// TIA Portal V19 export
FUNCTION_BLOCK "Prod_O_TODO_Push_ManualOrder"   // FB35, LAD
TITLE = INSERIMENTO MANAULE ORDINE SU LISTA ORDINI DA FARE (HMI -> TODO)
// stored: Access Published, MemoryReserve 100, SetENOAutomatically false
   VAR_INPUT
      Execute : Bool;
      Enable : Bool;
   END_VAR
   VAR_OUTPUT
      Ready : Bool;
      Busy : Bool;
      Done : Bool;
      Error : Bool;
   END_VAR
   VAR
      PPrf_Data_Presence { S7_SetPoint := 'True'} : Bool;
      WriteOrder : Bool;
      Prg { S7_SetPoint := 'True'} : "PPrf_Data";
      PPrf_Get { S7_SetPoint := 'True'} : "GetPrg";
      TON_Timeout { S7_SetPoint := 'True'} : TON_TIME;
      TON_Result { S7_SetPoint := 'True'} : TON_TIME;
      Order { S7_SetPoint := 'True'} : "Prod_Item";
      Counter_Space { S7_SetPoint := 'True'} : Int;
      RETVAL : DInt;
      TYP { ExternalAccessible := 'False'; ExternalVisible := 'False'; ExternalWritable := 'False'} : String;   // Tipo profilo (es. S, C)
      H_num : Real;
      H : String;
      W_num : Real;
      W : String;
      TK_num : Real;
      TK : String;
   END_VAR
   VAR_TEMP
      i : Int;
      Tol_Min : Real;
      Tol_Max : Real;
      Tol_Avg : Real;
      adj : Real;
   END_VAR
   VAR CONSTANT
      ERR_BEAMS_LEN : Int := -1;
      ERR_BEAM_REQ : Int := -2;
   END_VAR
   VAR_TEMP   // added for the SCL form of the ladder/FBD networks
      _w1 : Bool;
      _w2 : Bool;
   END_VAR
BEGIN

REGION Network 1: Reset stati precenti
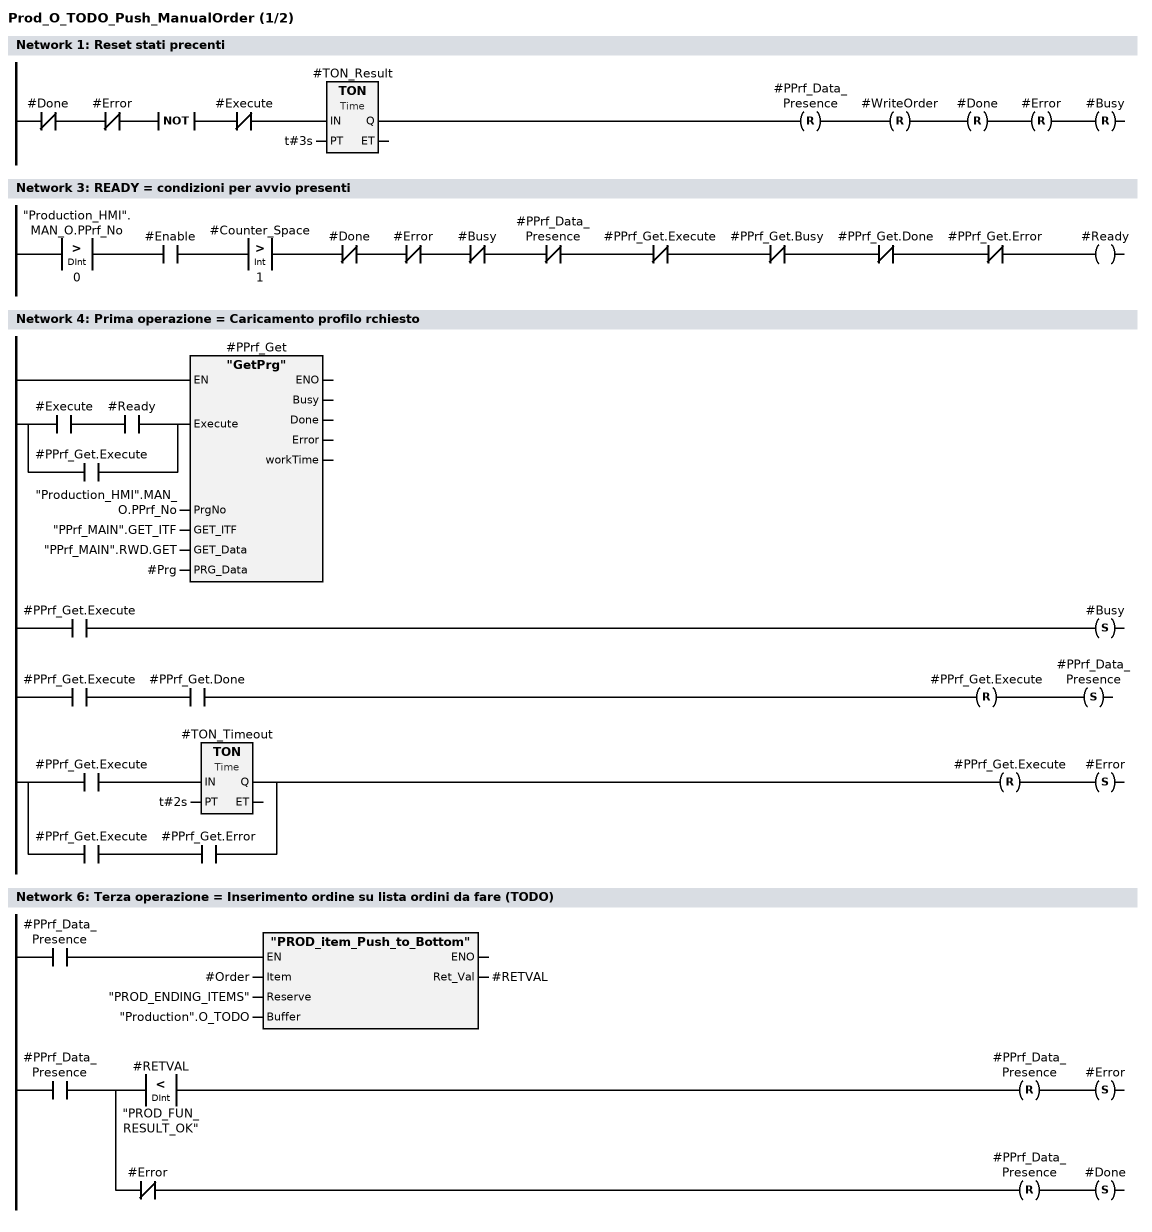
   RUNG wire#powerrail
      I_Contact( #Done )
      I_Contact( #Error )
      Not()
      I_Contact( #Execute )
      { S7_Templates := "time_type := Time" } #TON_Result.TON(pt := t#3s, et =>)
      R_Coil( #PPrf_Data_Presence )
      R_Coil( #WriteOrder )
      R_Coil( #Done )
      R_Coil( #Error )
      R_Coil( #Busy )
   END_RUNG
   // the same network as SCL:
   #TON_Result(IN := NOT (NOT #Done AND NOT #Error) AND NOT #Execute, PT := t#3s);   // TON
   IF #TON_Result.Q THEN
       #PPrf_Data_Presence := FALSE;
       #WriteOrder := FALSE;
       #Done := FALSE;
       #Error := FALSE;
       #Busy := FALSE;
   END_IF;
END_REGION

REGION Network 2 (SCL): Controlli preliminari sull'avvio eseguit se cìè abilitazione esterna e Profilo valorizzato
   IF "Production_HMI".MAN_O.PPrf_No > 0 AND #Enable THEN

       "Production_HMI".MAN_O.Req := MAX(IN1 := 1, IN2 := "Production_HMI".MAN_O.Req);


       "Production_HMI".MAN_O.Len := LIMIT_REAL(IN := "Production_HMI".MAN_O.Len, MN := "BEAM_LEN_MIN", MX := "BEAM_LEN_MAX");



       // Ricerca prima posizione libera
       // 

       #Counter_Space := 0;

       FOR #i := 1 TO "PROD_TODO_ITEMS" DO

           IF "Production".O_TODO[#i].O_ID <= 0 THEN
               #Counter_Space += 1;
           END_IF;

       END_FOR;
   END_IF;
END_REGION

REGION Network 3: READY = condizioni per avvio presenti
   RUNG wire#powerrail
      { S7_Templates := "SrcType := DInt" } GT_Contact(in1 := "Production_HMI".MAN_O.PPrf_No, in2 := 0)
      Contact( #Enable )
      { S7_Templates := "SrcType := Int" } GT_Contact(in1 := #Counter_Space, in2 := 1)
      I_Contact( #Done )
      I_Contact( #Error )
      I_Contact( #Busy )
      I_Contact( #PPrf_Data_Presence )
      I_Contact( #PPrf_Get.Execute )
      I_Contact( #PPrf_Get.Busy )
      I_Contact( #PPrf_Get.Done )
      I_Contact( #PPrf_Get.Error )
      Coil( #Ready )
   END_RUNG
   // the same network as SCL:
   #Ready := ("Production_HMI".MAN_O.PPrf_No > 0) AND #Enable AND (#Counter_Space > 1) AND NOT #Done AND NOT #Error AND NOT #Busy AND NOT #PPrf_Data_Presence AND NOT #PPrf_Get.Execute AND NOT #PPrf_Get.Busy AND NOT #PPrf_Get.Done AND NOT #PPrf_Get.Error;
END_REGION

REGION Network 4: Prima operazione = Caricamento profilo rchiesto
   RUNG wire#powerrail
      #PPrf_Get(Execute := wire#w1, PrgNo := "Production_HMI".MAN_O.PPrf_No, GET_ITF := "PPrf_MAIN".GET_ITF, GET_Data := "PPrf_MAIN".RWD.GET, PRG_Data := #Prg, Busy =>, Done =>, Error =>, workTime =>)
   END_RUNG
   RUNG wire#powerrail
      Contact( #Execute )
      Contact( #Ready )
   END_RUNG wire#w1
   RUNG wire#powerrail
      Contact( #PPrf_Get.Execute )
   END_RUNG wire#w1
   RUNG wire#powerrail
      Contact( #PPrf_Get.Execute )
      S_Coil( #Busy )
   END_RUNG
   RUNG wire#powerrail
      Contact( #PPrf_Get.Execute )
      Contact( #PPrf_Get.Done )
      R_Coil( #PPrf_Get.Execute )
      S_Coil( #PPrf_Data_Presence )
   END_RUNG
   RUNG wire#powerrail
      Contact( #PPrf_Get.Execute )
      { S7_Templates := "time_type := Time" } #TON_Timeout.TON(pt := t#2s, et =>)
      wire#w2
      R_Coil( #PPrf_Get.Execute )
      S_Coil( #Error )
   END_RUNG
   RUNG wire#powerrail
      Contact( #PPrf_Get.Execute )
      Contact( #PPrf_Get.Error )
   END_RUNG wire#w2
   // the same network as SCL:
   #PPrf_Get(Execute := (#Execute AND #Ready) OR #PPrf_Get.Execute,   // "GetPrg"
             PrgNo := "Production_HMI".MAN_O.PPrf_No,
             GET_ITF := "PPrf_MAIN".GET_ITF,
             GET_Data := "PPrf_MAIN".RWD.GET,
             PRG_Data := #Prg);
   IF #PPrf_Get.Execute THEN #Busy := TRUE; END_IF;
   #_w1 := #PPrf_Get.Execute AND #PPrf_Get.Done;
   IF #_w1 THEN
       #PPrf_Get.Execute := FALSE;
       #PPrf_Data_Presence := TRUE;
   END_IF;
   #TON_Timeout(IN := #PPrf_Get.Execute, PT := t#2s);   // TON
   #_w2 := #TON_Timeout.Q OR (#PPrf_Get.Execute AND #PPrf_Get.Error);
   IF #_w2 THEN
       #PPrf_Get.Execute := FALSE;
       #Error := TRUE;
   END_IF;
END_REGION

REGION Network 5 (SCL): Seconda operazione = Popolare dati dell'ordine
   IF #PPrf_Data_Presence AND NOT #WriteOrder THEN

       #WriteOrder := TRUE;

       #Order := "Production".O_Empty;


       #Order.O_ID := "Production".Last_O_ID + 1;


       #Order.Type := "PROD_ITEM_TYPE_HMI";

       #Order.MES_IDP := 'HMI';


       CASE #Prg.GeneralData.Beam_Code OF

           0:
               #Order.MES_Profile_Code := "PROFILE_TYPE_SEMIGUSCIO";


           1:
               #Order.MES_Profile_Code := "PROFILE_TYPE_ACCOPPIATO";
       END_CASE;

       #Order.MES_PPrf_Name := #Prg.Header.PrgName;


       #TYP := #Order.MES_Profile_Code;

       #H_num := INT_TO_REAL(#Prg.GeneralData.Beam_H_B_Code);

       #H := "Conv_NUM_to_STRING"(NumericValue := #H_num, NDec := 0);

       #W_num := INT_TO_REAL(#Prg.GeneralData.Beam_W_A_Code);

       #W := "Conv_NUM_to_STRING"(NumericValue := #W_num, NDec := 0);

       #TK_num := INT_TO_REAL(#Prg.GeneralData.Beam_TK_Code) / 100;

       #TK := "Conv_NUM_to_STRING"(NumericValue := #TK_num, NDec := 2);


       REGION FAKE PROFILE PROGRAM NAME BUILDING



           //--------------------------------------

           #Order.MES_PPrf_Name := '';


           #Order.MES_PPrf_Name := CONCAT(IN1 := #Order.MES_PPrf_Name, IN2 := #TYP);

           IF #H_num < 100 THEN

               #Order.MES_PPrf_Name := CONCAT(IN1 :=  #Order.MES_PPrf_Name, IN2 := '0');
           END_IF;

           #Order.MES_PPrf_Name := CONCAT(IN1 :=  #Order.MES_PPrf_Name, IN2 := #H);


           #Order.MES_PPrf_Name := CONCAT(IN1 :=  #Order.MES_PPrf_Name, IN2 := 'x');
           #Order.MES_PPrf_Name := CONCAT(IN1 :=  #Order.MES_PPrf_Name, IN2 := #W);


           #Order.MES_PPrf_Name := CONCAT(IN1 :=  #Order.MES_PPrf_Name, IN2 := 'x');
           #Order.MES_PPrf_Name := CONCAT(IN1 :=  #Order.MES_PPrf_Name, IN2 := #TK);

       END_REGION




       #Order.PPrf_No := "Production_HMI".MAN_O.PPrf_No;

       #Order.Beam_Code := #Prg.GeneralData.Beam_Code;
       #Order.Beams_W_A := #W_num;
       #Order.Beams_H_B := #H_num;
       #Order.Beams_Thickness :=#TK_num;

       #Order.Kanban_Style := FALSE;

       #Order.Use_Ribbing_Roll := "Production_HMI".MAN_O.Use_Ribbing_Roll;
       #Order.Use_Trace_Mark_Tool := "Production_HMI".MAN_O.Use_Trace_Mark_Tool;
       #Order.Use_Thick_Mark_Tool := "Production_HMI".MAN_O.Use_Thick_Mark_Tool;

       #Order.PackLayout_BeamsPerLayer := #Prg.GeneralData.PackLayout_BeamsPerLayer;
       #Order.PackLayout_Layers_Qty := #Prg.GeneralData.PackLayout_Layers_Qty;



       //@@@@@@@@@@@@@@@@@@@@@@@@@@@@@@@@@@@@@@@@@@@@@@@@@@@@@@@@@@
       // CALCOLO LUNGHEZZE MIN / MAX
       //@@@@@@@@@@@@@@@@@@@@@@@@@@@@@@@@@@@@@@@@@@@@@@@@@@@@@@@@@@ 

       #Order.Beams_Len := "Production_HMI".MAN_O.Len;



       #Tol_Min := "PLEN_TOL_MIN_DEFAULT";
       #Tol_Max := "PLEN_TOL_MAX_DEFAULT";

       IF (#Prg.GeneralData.Beam_Len_Tol_Max > #Prg.GeneralData.Beam_Len_Tol_Min)
           AND
           (#Prg.GeneralData.Beam_Len_Tol_Min <> 0.0 OR #Prg.GeneralData.Beam_Len_Tol_Max <> 0.0)
       THEN
           #Tol_Min := #Prg.GeneralData.Beam_Len_Tol_Min;
           #Tol_Max := #Prg.GeneralData.Beam_Len_Tol_Max;
       END_IF;

       #Order.Beams_Len_Min := #Order.Beams_Len + #Tol_Min;
       #Order.Beams_Len_Max := #Order.Beams_Len + #Tol_Max;

       #Tol_Avg := (#Tol_Max + #Tol_Min) / 2.0;

       #Order.Parts_Len := #Order.Beams_Len + #Tol_Avg;

       #Order.Parts_Tol := ABS(#Tol_Max - #Tol_Min) / 2.0;



       //@@@@@@@@@@@@@@@@@@@@@@@@@@@@@@@@@@@@@@@@@@@@@@@@@@@@@@@@@@
       // CONTATTORI PARTI / PEZZI
       //@@@@@@@@@@@@@@@@@@@@@@@@@@@@@@@@@@@@@@@@@@@@@@@@@@@@@@@@@@

       // Uscita con errore per quantità pezzi richiesta non valida
       // 

       #Order.Beams_REQ := "Production_HMI".MAN_O.Req;

       #Order.Beams_ToGo := #Order.Beams_REQ;


       #Order.Parts_REQ := #Order.Beams_REQ;

       IF #Order.Beam_Code = 1 THEN
           #Order.Parts_REQ := #Order.Parts_REQ * 2;
       END_IF;

       #Order.Parts_ToGo := #Order.Parts_REQ;


       //@@@@@@@@@@@@@@@@@@@@@@@@@@@@@@@@@@@@@@@@@@@@@@@@@@@@@@@@@@
       // QUANTITA' MATERIALE RICHIESTO
       //@@@@@@@@@@@@@@@@@@@@@@@@@@@@@@@@@@@@@@@@@@@@@@@@@@@@@@@@@@

       #Order.Material_Len_REQ := DINT_TO_REAL(#Order.Parts_REQ) * #Order.Parts_Len;
       #Order.Material_Len_ToGo := #Order.Material_Len_REQ;



   END_IF;
END_REGION

REGION Network 6: Terza operazione = Inserimento ordine su lista ordini da fare (TODO)
   RUNG wire#powerrail
      Contact( #PPrf_Data_Presence )
      "PROD_item_Push_to_Bottom"(Item := #Order, Reserve := "PROD_ENDING_ITEMS", Buffer := "Production".O_TODO, Ret_Val => #RETVAL)
   END_RUNG
   RUNG wire#powerrail
      Contact( #PPrf_Data_Presence )
      wire#w1
      { S7_Templates := "SrcType := DInt" } LT_Contact(in1 := #RETVAL, in2 := "PROD_FUN_RESULT_OK")
      R_Coil( #PPrf_Data_Presence )
      S_Coil( #Error )
   END_RUNG
   RUNG wire#w1
      I_Contact( #Error )
      R_Coil( #PPrf_Data_Presence )
      S_Coil( #Done )
   END_RUNG
   // the same network as SCL:
   IF #PPrf_Data_Presence THEN
       #RETVAL := "PROD_item_Push_to_Bottom"(Item := #Order,
                               Reserve := "PROD_ENDING_ITEMS",
                               Buffer := "Production".O_TODO);
   END_IF;
   #_w1 := #PPrf_Data_Presence AND (#RETVAL < "PROD_FUN_RESULT_OK");
   #_w2 := #PPrf_Data_Presence;
   IF #_w1 THEN
       #PPrf_Data_Presence := FALSE;
       #Error := TRUE;
   END_IF;
   IF #_w2 AND NOT #Error THEN
       #PPrf_Data_Presence := FALSE;
       #Done := TRUE;
   END_IF;
END_REGION

REGION Network 7: Quarta operazione = In caso di successo inizializza valori su HMI per prossimo inserimento
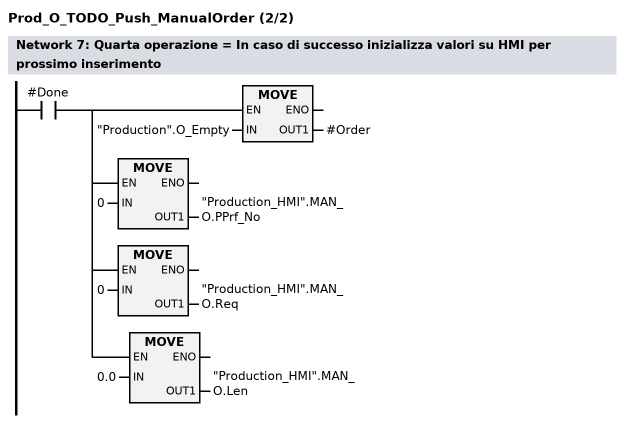
   RUNG wire#powerrail
      Contact( #Done )
      wire#w1
      Move(in := "Production".O_Empty, out1 => #Order)
   END_RUNG
   RUNG wire#w1
      { S7_GenerateENO := "TRUE" } Move(in := 0, out1 => "Production_HMI".MAN_O.PPrf_No)
   END_RUNG
   RUNG wire#w1
      { S7_GenerateENO := "TRUE" } Move(in := 0, out1 => "Production_HMI".MAN_O.Req)
   END_RUNG
   RUNG wire#w1
      { S7_GenerateENO := "TRUE" } Move(in := 0.0, out1 => "Production_HMI".MAN_O.Len)
   END_RUNG
   // the same network as SCL:
   IF #Done THEN
       #Order := "Production".O_Empty;
       "Production_HMI".MAN_O.PPrf_No := 0;
       "Production_HMI".MAN_O.Req := 0;
       "Production_HMI".MAN_O.Len := 0.0;
   END_IF;
END_REGION

REGION Network 8: +
END_REGION

REGION Network 9: +
END_REGION

REGION Network 10: +
END_REGION
END_FUNCTION_BLOCK
